// SIMATIC S7-200 project (STEP 7-Micro/WIN), CPU 224 REL 01.10

ORGANIZATION_BLOCK MAIN:OB1
TITLE=【【【【这个方案包含水泵控制和通讯模块，实现了住宅小区生活和消防两用水泵系统。】】】】
// 
// 系统运行的核心依赖于水源的可用性。
// 当水源信号为ON时，水源指示灯点亮，且系统允许水泵运行，但水泵启动需满足其他条件。
// 如果水源信号为OFF，系统会阻止水泵运行，以避免因无水源导致的空转损坏设备。
// 
// 
// 系统通过压力下限信号和压力上限信号实时监测水压。
// 当压力下限信号为ON或实时压力值低于设定值时，小流量泵启动延时定时器计时完成后置位小流量泵启动信号，点亮小流量泵运行指示灯，增加供水量。
// 如果小流量泵不足以满足需求，变频泵启动延时定时器2会进一步触发变频泵启动信号，通过变频泵选择信号决定启动一号水泵变频运行指示灯还是二号水泵变频运行指示灯。
// 反之，当压力上限信号为ON或实时压力值高于设定值时，小流量泵停止延时定时器或停泵延时定时器计时后停止相应水泵，确保水压始终维持在PID参数和压力设定值定义的范围内。
// 
// 
// 在水压持续偏低的情况下，加泵延时定时器会启动一号水泵工频运行指示灯或二号水泵工频运行指示灯，以工频模式增加供水能力；
// 当水压过高时，减泵延时定时器和减泵脉冲定时器协作置位减泵信号，逐步减少运行水泵数量。
// 第一恒压指示灯和第二恒压指示灯分别在不同运行状态下点亮，提示系统达到稳定的供水压力。
// 
// 系统安全性同样至关重要。
// 在自动模式下，若变频器故障信号为OFF且水源信号为ON，系统允许启动变频故障检测定时器（T37）以监测变频器状态。
// 当变频器故障信号为ON时，需确保一号水泵变频运行指示灯、二号水泵变频运行指示灯和小流量泵运行指示灯全部停止运行，点亮变频器故障指示灯，以保护设备和人员免受故障影响。
// 
// 
// 如果通讯状态标志异常或通讯故障标志置位，系统会暂停依赖通讯的操作，等待通讯恢复后再继续调整水泵状态，以保持供水过程的稳定性。
// 
// 
// 在手动模式下，操作员可通过小流量泵手动启动按钮、一号水泵手动启动按钮或二号水泵手动启动按钮直接控制水泵，手动加泵按钮和手动减泵按钮则通过手动加减泵延时定时器触发手动加减泵指示灯，灵活调整供水规模。
// 
// 
// 
BEGIN
Network 1 // 初始化
LD     SM0.1
CALL   SBR_0:SBR0            //初始化子程序
?000
Network 2
LDN    I0.0
O      M6.0
O      M6.2
O      M6.3
JMP    2
Network 3
LDW>=  VW176, +6
LPS
EU
CALL   SBR_10:SBR10
LPP
JMP    2
Network 4
LDB=   0, VB500
A      SM4.5
TON    T32, +20              //两次通讯之间时间间隔
Network 5
LD     T32
CALL   SBR_1:SBR1            //读变频器初值子程序
Network 6
LD     SM0.0
JMP    1
Network 7
LBL    2
//*******************定时读变频器参数*********************
Network 8 // 周期读实时频率及实时压力
LDB=   0, VB500
A      SM4.5
TON    T32, +20              //两次通讯之间的时间间隔
Network 9
LD     T32
CALL   SBR_2:SBR2            //读实时频率及实时压力参数子程序
//***********************运行程序**************************                                   
//KQK312BJ(A)-7.5KW运行程序
//I0.0 自动位 I0.1水源 I0.2变频故障 I0.3起动下限 I0.4起停上限
//Q0.0水源 Q0.1 1变 Q0.2 1工 Q0.3 2变 
//Q0.4 2工 Q0.5 小泵Q0.6 第一恒压 Q0.7第二恒压 Q1.0变频故障
Network 10
LD     I0.1
=      Q0.0                  //水源
Network 11
LDN    I0.2
O      M6.0
O      M6.1
O      M6.2
O      M6.3
O      M6.4
O      M6.5
A      I0.0
A      I0.1
TON    T37, +10
Network 12
LD     T37
=      M9.3                  //变频故障
R      Q3.1, 1
CALL   SBR_4:SBR4
Network 13
LD     I0.0
A      I0.1
LDW<=  VW44, VW6
O      I0.3                  //压力表下限
ALD
TON    T44, +30
Network 14
LD     T44
S      Q3.0, 1
Network 15
LDN    Q0.1
AN     Q0.3
A      I0.0
A      I0.1
AN     M9.3
A      Q3.0                  //小流量泵开
=      Q0.5
Network 16
LD     I0.4
OW>=   VW44, VW8             //压力表上限
AN     Q0.1
AN     Q0.3
A      I0.0
A      I0.1
TON    T38, +50
Network 17
LD     I0.0
A      I0.1
ED
O      T38
R      Q3.0, 1               //小流量泵停
Network 18
LD     Q0.5
AW<=   VW44, VW14
O      M9.5
TON    T39, +50
Network 19
LD     T39
A      I0.0
A      I0.1
S      Q3.1, 1               //变频泵运行
Network 20
LD     Q3.1
O      M9.0
O      M9.1
AN     M9.2
TON    T36, +5
Network 21
LD     T36
CALL   SBR_3:SBR3
Network 22
LD     Q0.1
O      Q0.3
AN     Q0.2
AN     Q0.4
AW>=   VW44, VW12
TON    T40, +150
Network 23
LD     I0.0
A      I0.1
ED
LD     T40
EU
OLD
R      Q3.1, 1               //变频器停止
CALL   SBR_4:SBR4
R      M9.5, 1
Network 24
LD     Q3.1
O      M9.0
O      M9.1
AN     M9.2
LPS
LD     Q0.1
ON     Q3.2
ALD                          //一变频运行 
AN     Q0.3
AN     M9.3
=      Q0.1
LPP
LD     Q0.3
O      Q3.2
ALD                          //二泵变频运行
AN     Q0.1
AN     M9.3
=      Q0.3
Network 25
LD     Q0.1
O      Q3.2
AN     Q0.3
=      Q3.2
Network 26
LD     Q0.1
O      Q0.3
A      I0.0
AN     M9.3
A      I0.1
AW<=   VW44, VW14
TON    T41, +100             //加泵信号
Network 27
LD     T41
O      Q0.2
O      Q0.4
AN     Q0.4
AN     Q3.3
A      Q0.3
LD     M9.3
AN     Q3.2
OLD
A      I0.0
A      Q0.0
=      Q0.2                  //一泵工频运行
Network 28
LD     T41
O      Q0.2
O      Q0.4
AN     Q0.2
AN     Q3.3
A      Q0.1
LD     M9.3
A      Q3.2
OLD
A      I0.0
A      Q0.0
=      Q0.4                  //二泵工频运行
Network 29
LD     Q0.1
A      Q0.4
LD     Q0.3
A      Q0.2
OLD
A      I0.0
A      I0.1
AN     M9.3
AW>=   VW44, VW16
TON    T42, +50              //减泵信号
Network 30
LD     T42
S      Q3.3, 1
Network 31
LD     Q3.3
TON    T43, +10              //1秒脉冲
Network 32
LD     T43
R      Q3.3, 1
Network 33
LD     Q0.1
O      Q0.3
AN     Q0.2
AN     Q0.4
O      T43
=      Q0.6                  //第一恒压
Network 34
LD     Q0.1
A      Q0.4
LD     Q0.3
A      Q0.2
OLD
O      Q3.3
=      Q0.7                  //第二恒压
Network 35
LD     I0.6
O      I0.7
TON    T50, +5
Network 36
// MEND
// 
LD     T50
=      M9.0
Network 37
LD     I1.1
O      M9.1
AN     I1.2
=      M9.1
Network 38
LD     Q0.1
ED
LD     Q0.3
ED
OLD
S      M9.2, 1
Network 39
LD     M9.2
TOF    T51, +100
Network 40
LD     T51
EU
R      M9.2, 1
Network 41
LD     M9.0
O      M9.1
=      Q1.1
Network 42
LD     Q0.2
AN     I0.3
LD     Q0.4
AN     I0.4
OLD
LD     Q0.5
AN     I0.5
OLD
A      I0.0
TON    T52, +20
Network 43
LD     T52
O      M9.3
S      Q1.0, 1
Network 44
LD     I0.0
A      I0.1
ED
R      Q1.0, 1
Network 45
LDN    Q0.2
AN     Q0.4
A      I1.0
S      M9.5, 1
Network 46
LBL    1
END_ORGANIZATION_BLOCK

SUBROUTINE_BLOCK SBR_0:SBR0
TITLE=
// *****************PORT0及变量初始化******************
// 
// 
BEGIN
Network 2
LD     SM0.0
MOVB   16#49, SMB30          //将PORT0设为自由口
//*******************POET0通讯区初始化***********************
MOVB   16#E, VB99            //LEN
MOVB   16#2, VB100           //STX
MOVB   16#C, VB101           //LGE
MOVB   0, VB102              //ADR
MOVW   +0, VW105             //IND
MOVW   +0, VW107             //VAL
MOVW   16#C7E, VW109         //STW
MOVW   +0, VW111             //HSW
Network 3
LD     SM0.0
FILL   +0, VW0, 20
FILL   +0, VW150, 25
MOVD   &VB0, VD150           //初始化接收地址指针
MOVW   +4, VW170             //通讯重试次数==VW170-1
MOVW   +6, VW172             //通讯允许连续出错次数==VW172-1
MOVW   +4, VW174             //变频故障允许重新启动重试次数==VW174-1
MOVW   +0, VW176
MOVB   0, VB500
R      M6.0, 8
Network 4
LD     SM0.0
MOVB   16#1, MB0
MOVB   16#FE, MB1
MOVB   16#0, MB2
Network 5
ENI                          //使中断使能
//******************PORT1通讯区初始化*************************
Network 6
//  RET
// 
END_SUBROUTINE_BLOCK

SUBROUTINE_BLOCK SBR_1:SBR1
TITLE=
// ******************读变频器初值子程序************************
// 
// 
BEGIN
Network 2 // 读P041
LDW=   +0, VW176
MOVW   16#1029, VW103        //PKE
JMP    0
Network 3 // 读P042
LDW=   +1, VW176
MOVW   16#102A, VW103
JMP    0
Network 4 // 读P043
LDW=   +2, VW176
MOVW   16#102B, VW103
JMP    0
Network 5 // 读P044
LDW=   +3, VW176
MOVW   16#102C, VW103
JMP    0
Network 6 // 读P046
LDW=   +4, VW176
MOVW   16#102E, VW103
JMP    0
Network 7 // 读P047
LDW=   +5, VW176
MOVW   16#102F, VW103
JMP    0
Network 8
LD     SM0.0
JMP    1
Network 9
LBL    0
Network 10
CALL   SBR_5:SBR5
CALL   SBR_6:SBR6
Network 11
LBL    1
Network 12
//  RET
// 
END_SUBROUTINE_BLOCK

SUBROUTINE_BLOCK SBR_2:SBR2
TITLE=**********************读P210及实时频率***********************
// 
BEGIN
Network 2
LD     SM0.0
MOVW   16#10D2, VW103
CALL   SBR_5:SBR5
CALL   SBR_8:SBR8
Network 3
//  RET
// 
END_SUBROUTINE_BLOCK

SUBROUTINE_BLOCK SBR_3:SBR3
TITLE=**********************启动变频器子程序************************
// 
BEGIN
Network 2
LD     SM0.0
MOVW   16#C7F, VW109
Network 3
//  RET
// 
END_SUBROUTINE_BLOCK

SUBROUTINE_BLOCK SBR_4:SBR4
TITLE=***********************停变频器子程序*************************
// 
BEGIN
Network 2
LD     SM0.0
MOVW   16#C7E, VW109
Network 3
//  RET
// 
END_SUBROUTINE_BLOCK

SUBROUTINE_BLOCK SBR_5:SBR5
TITLE=**********************运算BCC码子程序************************
// 
BEGIN
Network 2
LD     SM0.0
MOVB   0, VB113
MOVD   &VB100, AC1
Network 3
LD     SM0.0
FOR    AC3, +1, +13
XORB   *AC1, VB113
INCD   AC1
Network 4
NEXT
Network 5
//  RET
// 
END_SUBROUTINE_BLOCK

SUBROUTINE_BLOCK SBR_6:SBR6
TITLE=**************************发送子程序*************************
// 
BEGIN
Network 2
LD     SM0.0
XMT    VB99, 0
MOVB   16#FF, VB500
MOVB   100, SMB34
ATCH   INT_0:INT0, 9         //开PORT0发送结束中断
ATCH   INT_1:INT1, 10        //开PORT0发送超时中断
Network 3
//  RET
// 
END_SUBROUTINE_BLOCK

SUBROUTINE_BLOCK SBR_8:SBR8
TITLE=******************读实时频率及实时压力发送子程序**************
// 
BEGIN
Network 2
LD     SM0.0
XMT    VB99, 0
MOVB   16#FF, VB500
MOVB   100, SMB34
ATCH   INT_2:INT2, 9         //读实时频率及实时压力PORT0发送结束中断
ATCH   INT_3:INT3, 10        //读实时频率及实时压力PORT0超时中断
Network 3
//  RET
// 
END_SUBROUTINE_BLOCK

SUBROUTINE_BLOCK SBR_10:SBR10
TITLE=*******************PID上下限运算子程序************************
// 
BEGIN
Network 2
LD     SM0.0
MOVW   VW10, VW12
+I     VW0, VW12
MOVW   VW0, VW14
-I     VW10, VW14
MOVW   VW10, VW16
+I     VW2, VW16
MOVW   VW2, VW18
-I     VW10, VW18
MOVW   VW10, VW20
+I     VW4, VW20
MOVW   VW4, VW22
-I     VW10, VW22
MOVW   VW10, VW24
+I     VW6, VW24
MOVW   VW6, VW26
-I     VW10, VW26
MOVW   VW10, VW28
+I     VW8, VW28
MOVW   VW8, VW30
-I     VW10, VW30
Network 3
// RET
// 
END_SUBROUTINE_BLOCK

INTERRUPT_BLOCK INT_0:INT0
TITLE=******************PORT0发送结束中断程序***********************
// 
BEGIN
Network 2
LD     SM0.0
DTCH   10                    //退出XMT定时器
DTCH   9                     //终止XMT事件
MOVW   +14, VW180            //响应信息中接收的字符数
MOVB   0, VB190              //接收信息BCC码累加器
MOVD   &VB114, VD164         //设置接收缓冲区指针
MOVB   100, SMB34
ATCH   INT_4:INT4, 8         //开接收字符中断
ATCH   INT_5:INT5, 10        //开接受超时中断
Network 3
//  RETI
// 
END_INTERRUPT_BLOCK

INTERRUPT_BLOCK INT_1:INT1
TITLE=****************PORT0发送超时中断程序************************
// 
BEGIN
Network 2
LD     SM0.0
DTCH   9
DTCH   10
DECW   VW170
Network 3
LDW=   +0, VW170
EU
LPS                          //发送超时标志位
S      M6.0, 1
MOVB   3, VB192
MOVW   +4, VW170
MOVB   0, VB500
CRETI
NOT
A      SM4.5
XMT    VB99, 0
LRD
NOT
MOVB   16#FF, VB500
LRD
NOT
MOVB   100, SMB34
LRD
NOT
ATCH   INT_0:INT0, 9
LPP
NOT
ATCH   INT_1:INT1, 10
Network 4
//  RETI
// 
END_INTERRUPT_BLOCK

INTERRUPT_BLOCK INT_2:INT2
TITLE=************PORT0读实时频率及实时压力发送中断程序**************
// 
BEGIN
Network 2
LD     SM0.0
DTCH   9
DTCH   10
MOVW   +14, VW180            //接收字符数
MOVB   0, VB190              //BCC码累加器
MOVD   &VB114, VD164         //设置接收缓冲区地址指针
MOVB   100, SMB34
ATCH   INT_6:INT6, 8         //开接收中断
ATCH   INT_7:INT7, 10        //开接收超时中断
Network 3
//  RETI
// 
END_INTERRUPT_BLOCK

INTERRUPT_BLOCK INT_3:INT3
TITLE=**********PORT0读实时频率及实时压力发送超时中断程序*************
// 
BEGIN
Network 2
LD     SM0.0
DTCH   9
DTCH   10
MOVB   0, VB500
DECW   VW172
Network 3
LDW=   +0, VW172
S      M6.1, 1               //发送超时中断标志位
MOVW   +6, VW172
MOVB   3, VB192
Network 4
//  RETI
// 
END_INTERRUPT_BLOCK

INTERRUPT_BLOCK INT_4:INT4
TITLE=******************PORT0接收到字符中断************************
// 
BEGIN
Network 2
LD     SM0.0
MOVB   SMB2, AC0             //得到接收字符
XORB   AC0, VB190            //计算BCC码
MOVB   AC0, *VD164           //将接收字符送入缓冲区
INCD   VD164
DECW   VW180
Network 3
LDW=   +0, VW180
NOT
CRETI
Network 4
LD     SM0.0
DTCH   8
DTCH   10
MOVB   0, VB500              //接收结束允许再发送
AB=    0, VB190
NOT
MOVB   2, VB192
JMP    0
Network 5
LDB=   VB114, 16#2           //BCC码正确，检验其它部分]
AB=    VB115, 16#C
AB=    VB116, VB102
MOVW   +4, VW170             //刷新XMT重试次数==VW170-1
MOVB   0, VB192              //操作正确
MOVW   VW121, *VD150
INCD   VD150
INCD   VD150
INCW   VW176
JMP    1
Network 6
LD     SM0.0
MOVB   1, VB192              //信息中有不对的地方
Network 7
LBL    0
Network 8
LD     SM0.0
DECW   VW170
Network 9
LDW=   VW170, +0
LPS
NOT
MOVB   16#0, VB500
LPP
NOT
JMP    1
Network 10
LD     SM0.0
MOVW   +4, VW170
S      M6.2, 1               //接收字符出错标志位
Network 11
LBL    1
Network 12
//  RETI
// 
END_INTERRUPT_BLOCK

INTERRUPT_BLOCK INT_5:INT5
TITLE=*******************PORT0接收超时中断程序**********************
// 
BEGIN
Network 2
LD     SM0.0
DTCH   8
DTCH   10
MOVB   0, VB500
DECW   VW170
Network 3
LDW=   VW170, +0
MOVB   4, VB192
MOVW   +4, VW170
S      M6.3, 1               //接收字符超时故障标志位
CRETI
NOT
MOVB   16#0, VB500
Network 4
//  RETI
// 
END_INTERRUPT_BLOCK

INTERRUPT_BLOCK INT_6:INT6
TITLE=************读实时频率及实时压力接收字符中断程序**************
// 
BEGIN
Network 2
LD     SM0.0
MOVB   SMB2, AC0
XORB   AC0, VB190
MOVB   AC0, *VD164
INCD   VD164
DECW   VW180
Network 3
LDW=   VW180, +0
NOT
CRETI
Network 4
LD     SM0.0
DTCH   8
DTCH   10
MOVB   0, VB500
AB=    0, VB190
NOT
MOVB   2, VB192
JMP    0
Network 5
LDB=   VB114, 16#2
AB=    VB115, 16#C
AB=    VB116, VB102
R      M6.0, 6
MOVW   +6, VW172
MOVB   0, VB192
MOVW   +0, VW600             //计算实时频率
MOVW   VW125, VW602
MUL    +500, VD600
DTR    VD600, VD604
/R     16384.0, VD604
TRUNC  VD604, VD600
MOVW   VW602, VW46
MOVW   VW121, VW52           //计算实时压力（PID反馈值）
MOVW   +0, VW50
-D     +2000, VD50
DIV    +8, VD50
MOVW   VW52, VW44
JMP    1
NOT
MOVB   1, VB192
Network 6
LBL    0
Network 7
LD     SM0.0
MOVB   0, VB500
DECW   VW172
Network 8
LDW=   VW172, +0
MOVW   +6, VW172
S      M6.4, 1               //PORT0通讯连续出错标志位
Network 9
LBL    1
Network 10
LD     V22.7
MOVW   +0, VW22
Network 11
//  RETI
// 
END_INTERRUPT_BLOCK

INTERRUPT_BLOCK INT_7:INT7
TITLE=*************PORT0读实时频率及实时压力接收超时中断程序**************
// 
BEGIN
Network 2
LD     SM0.0
DTCH   8
DTCH   10
MOVB   0, VB500
DECW   VW172
Network 3
LDW=   VW172, +0
MOVW   +6, VW172
MOVB   4, VB192
S      M6.5, 1               //PORT0接收超时错误标志位
Network 4
//  RETI
// 
END_INTERRUPT_BLOCK
